TYPE Position :
STRUCT
	x : LREAL;	//Depth
	z : LREAL;	//Width
	y : LREAL;	//Height
END_STRUCT
END_TYPE

(* stored: Version 1.1.0.1, ProductVersion 3.1.4024.12
   DUT Position: Id {13aec421-2361-4438-b89d-cca6fca70b99} *)
